# EPICS substitutions: Db/waveform.substitutions
#Substitution file

file waveform.template
{
pattern
{channel}
{"0"}
{"1"}
{"2"}
  }
